// TIA Portal V19 export
DATA_BLOCK "SetPrfOnWork_IDB"   // DB21
// stored: InstanceOfName SetPrfOnWork, InstanceOfType FB
"SetPrfOnWork"
   // VAR_INPUT
   //    Enable : Bool;
   // END_VAR
   // VAR_IN_OUT
   //    HMI : "Prg_HMI";
   //    GET_ITF : "Prg_GetITF";
   //    GET_Data : Variant;
   //    PRG_Data : Variant;
   // END_VAR
   // VAR
   //    GetPrf : "GetPrg";
   //    tonDone { S7_SetPoint := 'True'} : IEC_TIMER;
   // END_VAR
BEGIN
END_DATA_BLOCK
